TYPE ST_ItemListOUT3 :
STRUCT
	ItemPK1 	:ST_ItemPK1_OUT3;
	ItemPK2 	:ST_ItemPK2_OUT3;
	ItemPK3 	:ST_ItemPK3_OUT3;
	ItemPK4 	:ST_ItemPK4_OUT3;
END_STRUCT
END_TYPE

(* stored: Version 1.1.0.1, ProductVersion 3.1.4024.13
   DUT ST_ItemListOUT3: Id {0d5f4437-96ae-453b-a08a-c025d027d6da} *)
